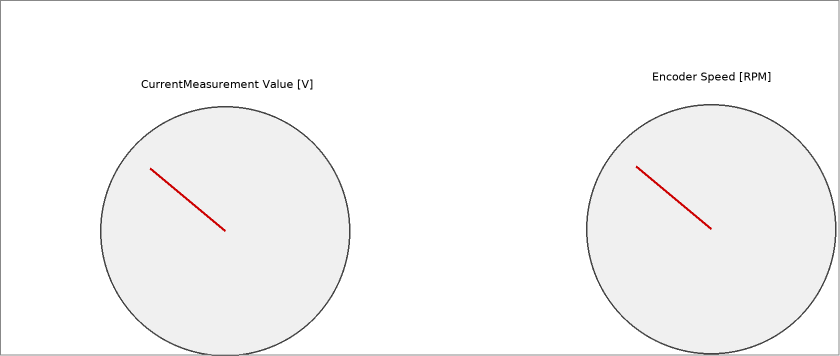
VISUALIZATION Visualization  // 840x356
    Meter180 (100,106 250x250), value: MAIN.CurrentMeasurement, style: Meter-Meter180-Gray, scale format: %.1f, scale -5..5
    Label (118,57 219x55), "CurrentMeasurement Value [V]"
    Meter180 (586,104 250x250), value: MAIN.CurrentMeasurement, style: Meter-Meter180-Gray, scale format: %.1f, scale 0..1000
    Label (584,47 256x60), "Encoder Speed [RPM]"
END_VISUALIZATION

(* stored: Version 1.1.0.1, ProductVersion 3.1.4024.11
   Visu Visualization: Id {106fe545-ae25-49e8-a5d3-8fa229086937} *)
